FUNCTION_BLOCK WARPPERSPECTIVE (* openCV warp perspective *)
  (* Version 1.0, AN, SWDC RTSoft *)
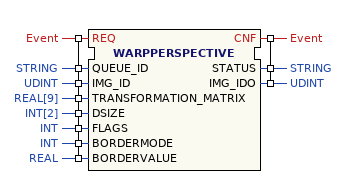
  EVENT_INPUT
    REQ WITH QUEUE_ID, IMG_ID, TRANSFORMATION_MATRIX, DSIZE, FLAGS, BORDERMODE, BORDERVALUE;
  END_EVENT
  EVENT_OUTPUT
    CNF WITH STATUS, IMG_IDO;
  END_EVENT
  VAR_INPUT
    QUEUE_ID : STRING;
    IMG_ID : UDINT;
    TRANSFORMATION_MATRIX : ARRAY [0..8] OF REAL; (* Array will be transformed into a 3x3 transformation matrix *)
    DSIZE : ARRAY [0..1] OF INT; (* Destination size [width, height] *)
    FLAGS : INT; (* 0: INTER_NEAREST, 1: INTER_LINEAR, 2: INTER_CUBIC, 3: INTER_AREA, 4: INTER_LANCZOS4 *)
    BORDERMODE : INT; (* 0: BORDER_CONSTANT, 1: BORDER_REPLICATE, 2: BORDER_REFLECT, 3: BORDER_WRAP, 4: BORDER_REFLECT_101, 5: BORDER_TRANSPARENT, 6: BORDER_REFLECT101, 7: BORDER_DEFAULT, 8: BORDER_ISOLATED *)
    BORDERVALUE : REAL;
  END_VAR
  VAR_OUTPUT
    STATUS : STRING;
    IMG_IDO : UDINT;
  END_VAR
  ALGORITHM REQ IN ST:

  END_ALGORITHM
END_FUNCTION_BLOCK
